FUNCTION_BLOCK ABSTRACT FB_Collection IMPLEMENTS I_Collection
VAR
	nCount 	: T_Capacity; // Size of Collection
	stError : T_Error := F_Error(FALSE, GVL_CmpErrors.ERR_OK,'');
END_VAR

(* Number of elements in collection*)
PROPERTY _Count : T_Capacity
GET
_Count := THIS^.nCount;
END_GET
END_PROPERTY

(* Gets collection's error status *)
PROPERTY _Error_Status : T_Error
GET
_Error_Status := THIS^.stError;
END_GET
SET // PROTECTED
THIS^.stError := THIS^.stError;
END_SET
END_PROPERTY

(* Checks if collection is empty.*)
PROPERTY _Is_Empty : BOOL
GET
_Is_Empty := THIS^._Count = 0;
END_GET
END_PROPERTY

(* Empties/Clears/Deletes every element on the collection*)
METHOD Clear
END_METHOD

METHOD PROTECTED ClearException : BOOL
VAR_INPUT
END_VAR
THIS^.stError := F_Error(FALSE, 0, '');
END_METHOD

// Clears value by setting it's entire memory space to NULL
METHOD PROTECTED ClearValue
VAR_INPUT
	Value : __SYSTEM.AnyType;
END_VAR
MEMSET(Value.pValue, 16#0, TO_UDINT(Value.diSize));
END_METHOD

// Copy data from source memory space to desination memory space
METHOD PROTECTED CopyValueTo
VAR_INPUT
	Dest, Src : __SYSTEM.AnyType;
END_VAR
THIS^.ClearValue(Dest);
MEMMOVE(Dest.pValue, Src.pValue, TO_UDINT(MIN(Dest.diSize, Src.diSize)));
END_METHOD

// Decrement list size by 1.
METHOD PROTECTED DecrementCount
VAR_INPUT
END_VAR
THIS^.nCount := THIS^.nCount - 1;
END_METHOD

// Raises an expection if list is empty
METHOD PROTECTED EmptyListException : BOOL
VAR_INPUT
END_VAR
IF THIS^._Is_Empty THEN THIS^.RaiseException(2936, 'Collection is empty'); EmptyListException := TRUE; END_IF
END_METHOD

METHOD PROTECTED FailedInsertionException : BOOL
VAR_INPUT
END_VAR
THIS^.RaiseException(2667, 'Failed to insert item into collection');
END_METHOD

// Increments list size by 1
METHOD PROTECTED IncrementCount
VAR_INPUT
END_VAR
THIS^.nCount := THIS^.nCount + 1;
END_METHOD

METHOD PROTECTED NullReferenceException : BOOL
THIS^.RaiseException(2000+GVL_CmpErrors.ERR_INVALID_REFERENCE, 'Null or Invalid Reference');
END_METHOD

METHOD PROTECTED OutOfBoundsException : BOOL
VAR_INPUT
	nIndex : T_Capacity;
END_VAR
IF (nIndex < 0) OR (nIndex >= THIS^._Count) THEN
	THIS^.RaiseException(2374,'Out of bounds. You tried to access data outside the range of this collection.');
	OutOfBoundsException := TRUE;
	END_IF
END_METHOD

METHOD PROTECTED RaiseException : BOOL
VAR_INPUT
	nCode 	: DINT;
	sSource : T_MaxString;
END_VAR
THIS^.stError := F_Error(TRUE, nCode, sSource);
END_METHOD

METHOD PROTECTED ValueFoundException : BOOL
VAR_INPUT
END_VAR
THIS^.RaiseException(2748, 'Value is contained in collection');
END_METHOD

METHOD PROTECTED ValueNotFoundException : BOOL
VAR_INPUT
END_VAR
THIS^.RaiseException(2923, 'Value is not contain in collection');
END_METHOD

END_FUNCTION_BLOCK

(* stored: Version 1.1.0.1, ProductVersion 3.1.4024.4
   POU FB_Collection: Id {8169983e-4d36-41ab-8620-a5d13bfe975a}, SpecialFunc None
   Folder Exception Handling: Id {e863efaf-051a-44d3-96d3-01058ddc780e}
   Folder Protected: Id {8019ce0d-62b9-4c90-857c-02dfeaf35f02}
   Property _Count: Id {6000edd3-5a9e-4b73-8290-ee5244a090cf}
   Get Get: Id {90d08fe7-41c4-4166-8944-ea4694f441f8}
   Property _Error_Status: Id {cf5de7bc-ad33-4e64-8887-853375cfc8c8}
   Get Get: Id {8db0a8ee-7feb-438f-be99-f72530da82d2}
   Set Set: Id {fa4af9d6-43ec-4e3e-bdcd-c88b0dd4815e}
   Property _Is_Empty: Id {9745dabf-5a07-43e1-acf4-a7a1da3163d9}
   Get Get: Id {a8515034-4356-4e11-aa1b-c1ea197c4dff}
   Method Clear: Id {cb80021a-e4cc-4394-bdef-8b703b603d7f}
   Method ClearException: Id {fa6fc6d6-d879-49f9-9bc2-01521bc9012c}
   Method ClearValue: Id {c5c5bce6-4d81-43ca-9908-7dd2ab56be33}
   Method CopyValueTo: Id {56538ce5-958a-4337-bfb7-cab401b0c3a6}
   Method DecrementCount: Id {cbc4706b-c46f-41a4-a1a1-d47131fab88c}
   Method EmptyListException: Id {e5e86fcd-94fa-4e43-bc44-9673d72b84e8}
   Method FailedInsertionException: Id {e5949954-ed95-4829-b875-1dc2e716e1f9}
   Method IncrementCount: Id {88677d6e-fe73-41cf-a02d-1dd614bad8d5}
   Method NullReferenceException: Id {6929719b-42b1-49b7-b2d4-2fdc2342d4cc}
   Method OutOfBoundsException: Id {29cc68fc-ef87-48b1-a4ed-8dcabf95dcfe}
   Method RaiseException: Id {a53dccc9-6cca-4cc6-96bd-709718fb0e6a}
   Method ValueFoundException: Id {f14aa7ba-deb7-4a2e-9f77-7c1a41907382}
   Method ValueNotFoundException: Id {55c2a48e-7f84-4826-b079-cdf74763177e} *)
